// TIA Portal project "2022.04.24-S和R" (V17)

(* hardware
DEVICE "S7-1500/ET200MP station_1"  S7-1500 station
   slot 0: "导轨_0"  Rack  6ES7 590-1***0-0AA0
   slot 1: "PLC_1"  CPU 1516-3 PN/DP  6ES7 516-3AN00-0AB0  V1.7
      slot 3: "CPU 显示_1"  6ES7591-1BA00-0AA0
      slot 32768: "PROFINET 接口_1"  X1
         slot 32769: "端口_1"  X1 P1
         slot 32770: "端口_2"  X1 P2
      slot 33024: "PROFINET 接口_2"  X2
         slot 33025: "端口_1"  X2 P1
      slot 33280: "DP 接口_1"  X3
   slot 2: "DI 32x24VDC BA_1"  DI 32x24VDC BA  6ES7 521-1BL10-0AA0  V1.1
   slot 3: "DQ 32x24VDC/0.5A HF_1"  DQ 32x24VDC/0.5A HF  6ES7 522-1BL01-0AB0  V1.1
*)

// ===== PLC "PLC_1"  CPU 1516-3 PN/DP =====

VAR_GLOBAL   // PLC tag table "默认变量表"
   "按钮1" AT %I0.0 : Bool;
   "按钮2" AT %I0.1 : Bool;
   "按钮3" AT %I0.2 : Bool;
   "按钮4" AT %I0.3 : Bool;
   "按钮5" AT %I0.4 : Bool;
   "按钮6" AT %I0.5 : Bool;
   "按钮7" AT %I0.6 : Bool;
   "按钮8" AT %I0.7 : Bool;
   "按钮9" AT %I1.0 : Bool;
   "按钮10" AT %I1.1 : Bool;
   "按钮11" AT %I1.2 : Bool;
   "指示灯1" AT %Q0.0 : Bool;
   "指示灯2" AT %Q0.1 : Bool;
   "指示灯3" AT %Q0.2 : Bool;
   "指示灯4" AT %Q0.3 : Bool;
   "指示灯5" AT %Q0.4 : Bool;
   "指示灯6" AT %Q0.5 : Bool;
   "指示灯7" AT %Q0.6 : Bool;
   "指示灯8" AT %Q0.7 : Bool;
   "指示灯9" AT %Q1.0 : Bool;
   "指示灯10" AT %Q1.1 : Bool;
   "指示灯11" AT %Q1.2 : Bool;
   "指示灯12" AT %Q1.3 : Bool;
END_VAR

FUNCTION "置位与复位" : Void   // FC1, LAD
{ S7_Optimized_Access := 'TRUE' }
VERSION : 0.1
BEGIN

REGION Network 1
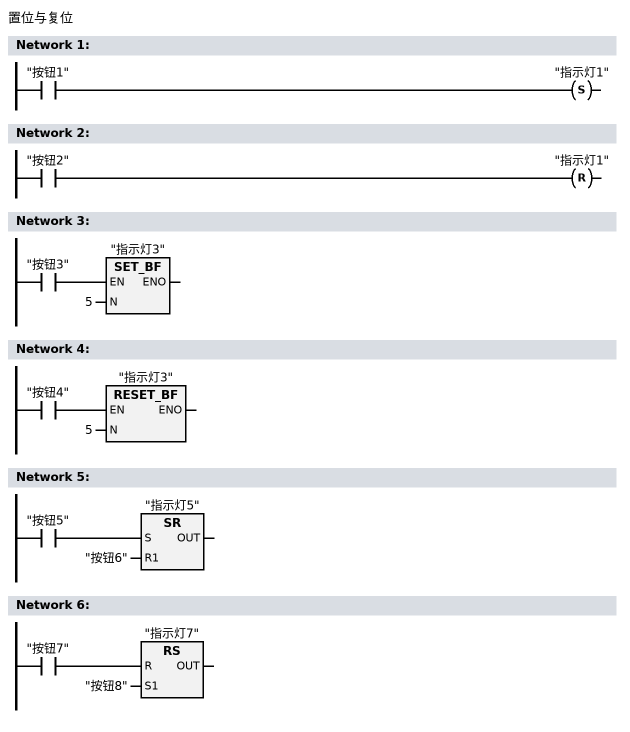
   RUNG wire#powerrail
      Contact( "按钮1" )
      S_Coil( "指示灯1" )
   END_RUNG
   // the same network as SCL:
   IF "按钮1" THEN "指示灯1" := TRUE; END_IF;
END_REGION

REGION Network 2
   RUNG wire#powerrail
      Contact( "按钮2" )
      R_Coil( "指示灯1" )
   END_RUNG
   // the same network as SCL:
   IF "按钮2" THEN "指示灯1" := FALSE; END_IF;
END_REGION

REGION Network 3
   // no SCL statement known for SBitfield: written as a call
   IF "按钮3" THEN SET_BF(operand := "指示灯3", n := 5); END_IF;
END_REGION

REGION Network 4
   // no SCL statement known for RBitfield: written as a call
   IF "按钮4" THEN RESET_BF(operand := "指示灯3", n := 5); END_IF;
END_REGION

REGION Network 5
   RUNG wire#powerrail
      Contact( "按钮5" )
      S_SR(operand := "指示灯5", r1 := "按钮6")
   END_RUNG
   // the same network as SCL:
   IF "按钮5" THEN
       "指示灯5" := TRUE;   // SR flip-flop
   END_IF;
   IF "按钮6" THEN "指示灯5" := FALSE; END_IF;
END_REGION

REGION Network 6
   RUNG wire#powerrail
      Contact( "按钮7" )
      S_RS(operand := "指示灯7", s1 := "按钮8")
   END_RUNG
   // the same network as SCL:
   IF "按钮7" THEN
       "指示灯7" := FALSE;   // RS flip-flop
   END_IF;
   IF "按钮8" THEN "指示灯7" := TRUE; END_IF;
END_REGION
END_FUNCTION

FUNCTION "置位复位FBD" : Void   // FC2, FBD
{ S7_Optimized_Access := 'TRUE' }
VERSION : 0.1
   VAR_TEMP   // added for the SCL form of the ladder/FBD networks
      _w1 : Bool;
   END_VAR
BEGIN

REGION Network 1
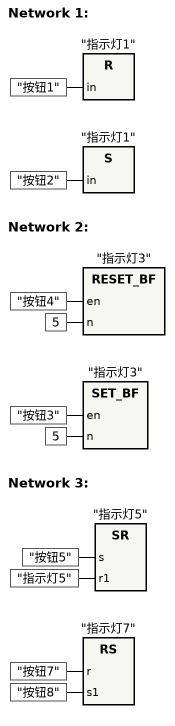
   IF "按钮1" THEN "指示灯1" := FALSE; END_IF;
   IF "按钮2" THEN "指示灯1" := TRUE; END_IF;
END_REGION

REGION Network 2
   // no SCL statement known for RBitfield, SBitfield: written as a call
   IF "按钮4" THEN RESET_BF(operand := "指示灯3", n := 5); END_IF;
   IF "按钮3" THEN SET_BF(operand := "指示灯3", n := 5); END_IF;
END_REGION

REGION Network 3
   #_w1 := "指示灯5";
   IF "按钮5" THEN
       "指示灯5" := TRUE;   // SR flip-flop
   END_IF;
   IF #_w1 THEN "指示灯5" := FALSE; END_IF;
   IF "按钮7" THEN
       "指示灯7" := FALSE;   // RS flip-flop
   END_IF;
   IF "按钮8" THEN "指示灯7" := TRUE; END_IF;
END_REGION
END_FUNCTION

FUNCTION "置位与复位SCL" : Void   // FC3, SCL
{ S7_Optimized_Access := 'TRUE' }
VERSION : 0.1
BEGIN
   IF "按钮1" THEN
       // Statement section IF
       "指示灯1":=FALSE
       ;
   END_IF;
   IF "按钮2" THEN
       // Statement section IF
       "指示灯1" := TRUE
       ;
   END_IF;


   //模拟置位域复位域
   IF "按钮3" THEN
       // Statement section IF
       "指示灯3" := TRUE;
       "指示灯4" := TRUE;
       "指示灯5" := TRUE;
       "指示灯6" := TRUE;
       "指示灯7" := TRUE
       ;
   END_IF;
   IF "按钮4" THEN
       // Statement section IF
       "指示灯3" := FALSE;
       "指示灯4" := FALSE;
       "指示灯5" := FALSE;
       "指示灯6" := FALSE;
       "指示灯7" := FALSE
       ;
   END_IF;
END_FUNCTION

ORGANIZATION_BLOCK "Main"   // OB1, LAD, ProgramCycle
TITLE = "Main Program Sweep (Cycle)"
{ S7_Optimized_Access := 'TRUE' }
VERSION : 0.1
   VAR_INPUT
      Initial_Call : Bool;   // Initial call of this OB
      Remanence : Bool;   // =True, if remanent data are available
   END_VAR
BEGIN

REGION Network 1
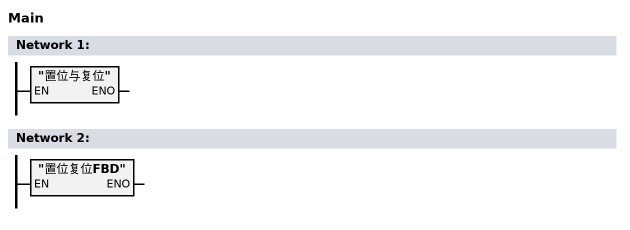
   RUNG wire#powerrail
      "置位与复位"()
   END_RUNG
   // the same network as SCL:
   "置位与复位"();
END_REGION

REGION Network 2
   RUNG wire#powerrail
      "置位复位FBD"()
   END_RUNG
   // the same network as SCL:
   "置位复位FBD"();
END_REGION
END_ORGANIZATION_BLOCK